INTERFACE IPAMSilo EXTENDS IPAProcessModule

END_INTERFACE

(* stored: Version 1.1.0.1, ProductVersion 3.1.4020.12
   Itf IPAMSilo: Id {9a3a86b7-83e7-4aae-b877-c68cfa3e4fe7} *)
